FUNCTION_BLOCK PUBLIC FB_DevAnalogAxis EXTENDS FB_DevBase
VAR_INPUT
	stManualCtrl 	: ST_ManualAnalogAxisCtrl ; // Manual control
END_VAR
VAR_OUTPUT
	bDriveOk		: BOOL ; // Drive is ok
	bMovingCW		: BOOL ; // Move CW output is active
	bMovingCCW		: BOOL ; // Move CCW output is active
	fActVelocity	: LREAL; // Command velocity of motor
END_VAR
VAR // internal functions 
	fbVelocity		: FB_DevAnalogOutputScaled 	;
	fbqRun			: FB_DevDigitalOutput		;
	fbqReset		: FB_DevDigitalOutput		;
	fbqReverse		: FB_DevDigitalOutput		;
	fbiEnabled		: Fb_DevDigitalInput		;
END_VAR
VAR // Internal commands
	fCmdVelocity	: LREAL;
	bCmdRunCW 		: BOOL ;
	bCmdRunCCW		: BOOL ;
	bCmdReset		: BOOL ;	 
	bInternalEnable : BOOL ;
END_VAR

SUPER^(refFbFault := refFbFault);

// ===== Check inputs =====
	fbiEnabled( bEmbeded	:= TRUE,
				refFbFault 	:= refFbFault);

IF bInitOk THEN 
	ExecSetOutputs() ;
	bDriveOk	:= fbiEnabled.bFcoInputActive ;
END_IF

METHOD PUBLIC CmdManual : BOOL
VAR_INPUT
END_VAR
bCmdManual := TRUE ;

// Execute Manual commands
	IF stManualCtrl.bCmdRunCW THEN 
		CmdRunCW(fCmdVelocity := stManualCtrl.fCmdVelocity);
	ELSIF stManualCtrl.bCmdRunCCW THEN 
		CmdRunCCW(fCmdVelocity := stManualCtrl.fCmdVelocity);
	END_IF
END_METHOD

METHOD PUBLIC CmdReset : BOOL
VAR_INPUT
END_VAR
bErrorActive 	:= FALSE;

bCmdReset		:= TRUE ;

CmdReset		:= TRUE ;
END_METHOD

METHOD PUBLIC CmdRunCCW : BOOL
VAR_INPUT
	fCmdVelocity	: LREAL ; // Command velocity
END_VAR
bCmdRunCCW			:= TRUE ;
THIS^.fCmdVelocity 	:= fCmdVelocity ; 

CmdRunCCW 	:= bMovingCW ;
END_METHOD

METHOD PUBLIC CmdRunCW : BOOL
VAR_INPUT
	fCmdVelocity	: LREAL ; // Command velocity
END_VAR
bCmdRunCW := TRUE ;
THIS^.fCmdVelocity 	:= fCmdVelocity ;

CmdRunCW 	:= bMovingCW ;
END_METHOD

METHOD PUBLIC CmdSafeStop : BOOL
VAR_INPUT
END_VAR
bIsSafe := TRUE ;

bIsSafe := fbVelocity.CmdSafeStop() AND bIsSafe ;
bIsSafe := fbqRun.CmdSafeStop() 	AND bIsSafe ;
bIsSafe := fbqReverse.CmdSafeStop() AND bIsSafe ;
bIsSafe := fbqReset.CmdSafeStop() 	AND bIsSafe ;

CmdSafeStop := bIsSafe;
END_METHOD

METHOD PRIVATE ExecSetOutputs : BOOL
VAR_INPUT
END_VAR
// ====== Check safety and enable ======
IF bSafetyOk 
AND fbiEnabled.bFcoInputActive 
AND (bEnable OR bManual) THEN 
	bInternalEnable := TRUE;
ELSE
	fCmdVelocity 	:= 0;
	bCmdRunCW		:= FALSE;
	bCmdRunCCW		:= FALSE;
END_IF 

{warning disable C0371}
// ====== Set outputs =======
	fbVelocity	(	bEmbeded 	:= TRUE,
					bSafetyOk	:= bSafetyOk,
					bEnable		:= bInternalEnable,
					fCmdValue	:= fCmdVelocity, 
					refFbFault	:= refFbFault);
				
	fbqRun		(	bEmbeded 	:= TRUE,
					bSafetyOk	:= bSafetyOk,
					bEnable		:= bInternalEnable,
					bCmdOn		:= bCmdRunCW OR bCmdRunCCW,
					refFbFault	:= refFbFault);
				
	fbqReverse	(	bEmbeded 	:= TRUE,
					bSafetyOk	:= bSafetyOk,
					bEnable		:= bInternalEnable,
					bCmdOn		:= bCmdRunCCW,
					refFbFault	:= refFbFault);

	fbqReset	(	bEmbeded 	:= TRUE,
					bSafetyOk	:= bSafetyOk,
					bEnable		:= bInternalEnable,
					bCmdOn		:= bCmdReset,
					refFbFault	:= refFbFault);
{warning restore C0371}
// ===== reset input commands =====
	fCmdVelocity 	:= 0;
	bCmdRunCW		:= FALSE;
	bCmdRunCCW		:= FALSE;
	bCmdManual		:= FALSE;
	bCmdReset		:= FALSE;
	bInternalEnable := FALSE;
// ===== set feedback =====

bMovingCW		:= fbqRun.bOutputState AND NOT fbqReverse.bOutputState;
bMovingCCW		:= fbqRun.bOutputState AND fbqReverse.bOutputState;
fActVelocity	:= fbVelocity.fOutputValue ;
END_METHOD

METHOD Init : BOOL
VAR_INPUT
	// Message location data
	nId			: UDINT ; // Identification number of object
	nParentId	: UDINT ; // Id of higher level If aplicable (0 = no parent)

	// Motor settings
	fMaxVelocity : LREAL ; // Maximum motor velocity for scaling
END_VAR
// ====== initialize components =====
	bInitOk := TRUE ;

// ====== Calculate device id =====
	bInitOk :=	ExecIdentifyDevice(nId,nParentId, E_ComponentTypes.Axis) AND bInitOk;

// ====== Set manual device type ======
	eDevType := E_Devices.AnalogAxis ;	


bInitOk := 	fbVelocity.Init	( 	nId 			:= 0,
								nParentId		:= nLocationId,
								benableNegative	:= FALSE )
								AND bInitOk;
			fbVelocity.SetScaling	(fMaxValue 		:= fMaxVelocity);
								
bInitOk	:= 	fbqRun.Init		( 	nId				:= 1,
								nParentId		:= nLocationId)
								AND bInitOk;

bInitOk	:= 	fbqReset.Init	( 	nId				:= 2,
								nParentId		:= nLocationId)
								AND bInitOk;

bInitOk	:= 	fbqReverse.Init	( 	nId				:= 3,
								nParentId		:= nLocationId)
								AND bInitOk;

bInitOk	:= 	fbiEnabled.Init	( 	nId				:= 4,
								nParentId		:= nLocationId)
								AND bInitOk;

// ====== Set feedback =======
Init := bInitOk;
END_METHOD

END_FUNCTION_BLOCK

(* stored: Version 1.1.0.1, ProductVersion 3.1.4024.10
   POU FB_DevAnalogAxis: Id {2d577320-0726-040c-269d-52c0e83d50e7}, SpecialFunc None
   Folder Commands: Id {25bd60d6-a0c4-006b-1e1e-40f55b890b42}
   Folder Private: Id {a644719c-3261-0f8c-3b05-3c6242d33819}
   Method CmdManual: Id {d526230f-e04e-08a3-0a52-d542f08f92a4}
   Method CmdReset: Id {69edc11b-9665-0aa5-3d5e-a0ff9e474fd0}
   Method CmdRunCCW: Id {e92c1c28-51a1-0de5-0174-155a52f08ed3}
   Method CmdRunCW: Id {e890e9f0-dd77-0270-3233-14c16580ad18}
   Method CmdSafeStop: Id {c1b9e61f-17d6-00f9-1428-4bb1000131d5}
   Method ExecSetOutputs: Id {73c3f618-cb9e-0650-0e12-802c6dbad778}
   Method Init: Id {1d9ecc1b-c37a-0e07-3bc6-88c35083f504} *)
